TYPE ST_OperationVars_DCcharger :
STRUCT
	b_StartCharging						: BOOL;
	b_ResetCharger						: BOOL;
END_STRUCT
END_TYPE

(* stored: Version 1.1.0.1, ProductVersion 3.1.4026.18
   DUT ST_OperationVars_DCcharger: Id {ebf75300-ce10-4eba-b2ae-a1ea8729d45f} *)
